// TIA Portal V17 export
// export: Created 2026-04-13T11:12:53.5499965Z, ExportSetting WithDefaults, DisplayName Totally Integrated Automation Portal, DisplayVersion V17 Update 4, DisplayName TIA Portal Openness, DisplayVersion V17 Update 4, DisplayName TIA Portal Version Control Interface, DisplayVersion V17, DisplayName SINAMICS Startdrive Advanced, DisplayVersion V17, DisplayName SINAMICS Startdrive G130, G150, S120, S150, SINAMICS MV, S210, DisplayVersion V17, DisplayName SINAMICS Startdrive G110M, G120, G120C, G120D, G120P, G115D, DisplayVersion V17, DisplayName STEP 7 Professional, DisplayVersion V17 Update 4, DisplayName STEP 7 Safety, DisplayVersion V17, DisplayName WinCC Professional, DisplayVersion V17 Update 4
TagTable "M"
  MABQ进水隔断阀 : Bool  (PLC tag MABQ进水隔断阀, HMI_连接_1, 1 s)
  MAB进水隔断阀 : Bool  (PLC tag MAB进水隔断阀, HMI_连接_1, 1 s)
  MAQ安全停机 : Bool  (PLC tag MAQ安全停机, HMI_连接_1, 1 s)
  MAS室内回水阀 : Bool  (PLC tag MAS室内回水阀, HMI_连接_1, 1 s)
  MAS室外回水阀 : Bool  (PLC tag MAS室外回水阀, HMI_连接_1, 1 s)
  MBD本地调试 : Bool  (PLC tag MBD本地调试, HMI_连接_1, 1 s)
  MBD补氮阀 : Bool  (PLC tag MBD补氮阀, HMI_连接_1, 1 s)
  MBD布袋出料 : Bool  (PLC tag MBD布袋出料, HMI_连接_1, 1 s)
  MBJ本机调试模式 : Bool  (PLC tag MBJ本机调试模式, HMI_连接_1, 1 s)
  MBS闭式进风隔断阀 : Bool  (PLC tag MBS闭式进风隔断阀, HMI_连接_1, 1 s)
  MBS闭式排风隔断阀 : Bool  (PLC tag MBS闭式排风隔断阀, HMI_连接_1, 1 s)
  MBY100 : Bool  (PLC tag MBY100, HMI_连接_1, 1 s)
  MBY101 : Bool  (PLC tag MBY101, HMI_连接_1, 1 s)
  MCC除尘出料上阀 : Bool  (PLC tag MCC除尘出料上阀, HMI_连接_1, 1 s)
  MCC除尘出料下阀 : Bool  (PLC tag MCC除尘出料下阀, HMI_连接_1, 1 s)
  MCC除尘管道清洗阀 : Bool  (PLC tag MCC除尘管道清洗阀, HMI_连接_1, 1 s)
  MCC除尘缓存震荡器 : Bool  (PLC tag MCC除尘缓存震荡器, HMI_连接_1, 1 s)
  MCC除尘脉冲 : Bool  (PLC tag MCC除尘脉冲, HMI_连接_1, 1 s)
  MCC除尘气锤 : Bool  (PLC tag MCC除尘气锤, HMI_连接_1, 1 s)
  MCC除尘清洗阀 : Bool  (PLC tag MCC除尘清洗阀, HMI_连接_1, 1 s)
  MCF出风高效清洗阀 : Bool  (PLC tag MCF出风高效清洗阀, HMI_连接_1, 1 s)
  MCS纯水洗请求 : Bool  (PLC tag MCS纯水洗请求, HMI_连接_1, 1 s)
  MCW除雾排液阀 : Bool  (PLC tag MCW除雾排液阀, HMI_连接_1, 1 s)
  MCZ初状态 : Bool  (PLC tag MCZ初状态, HMI_连接_1, 1 s)
  MDJ电加热器 : Bool  (PLC tag MDJ电加热器, HMI_连接_1, 1 s)
  MEJ二级出料 : Bool  (PLC tag MEJ二级出料, HMI_连接_1, 1 s)
  MEJ二级出料上阀 : Bool  (PLC tag MEJ二级出料上阀, HMI_连接_1, 1 s)
  MEJ二级出料下阀 : Bool  (PLC tag MEJ二级出料下阀, HMI_连接_1, 1 s)
  MEJ二级缓存震荡器 : Bool  (PLC tag MEJ二级缓存震荡器, HMI_连接_1, 1 s)
  MEJ二级冷冻水阀 : Bool  (PLC tag MEJ二级冷冻水阀, HMI_连接_1, 1 s)
  MEJ二级冷凝清洗阀 : Bool  (PLC tag MEJ二级冷凝清洗阀, HMI_连接_1, 1 s)
  MEJ二级排液阀 : Bool  (PLC tag MEJ二级排液阀, HMI_连接_1, 1 s)
  MEJ二级旋风气锤 : Bool  (PLC tag MEJ二级旋风气锤, HMI_连接_1, 1 s)
  MEJ二级旋风清洗阀 : Bool  (PLC tag MEJ二级旋风清洗阀, HMI_连接_1, 1 s)
  MEJ二级旋风振打锤 : Bool  (PLC tag MEJ二级旋风振打锤, HMI_连接_1, 1 s)
  MFK放空比例调节阀 : Bool  (PLC tag MFK放空比例调节阀, HMI_连接_1, 1 s)
  MFM蜂鸣器 : Bool  (PLC tag MFM蜂鸣器, HMI_连接_1, 1 s)
  MFZ仿真调试 : Bool  (PLC tag MFZ仿真调试, HMI_连接_1, 1 s)
  MGD管道压力手动调节 : Bool  (PLC tag MGD管道压力手动调节, HMI_连接_1, 1 s)
  MGS供水泵 : Bool  (PLC tag MGS供水泵, HMI_连接_1, 1 s)
  MHF回风加热比例调节阀 : Bool  (PLC tag MHF回风加热比例调节阀, HMI_连接_1, 1 s)
  MHF回风加热自整定 : Bool  (PLC tag MHF回风加热自整定, HMI_连接_1, 1 s)
  MHF回风温度加热 : Bool  (PLC tag MHF回风温度加热, HMI_连接_1, 1 s)
  MHF回风蒸汽开关阀 : Bool  (PLC tag MHF回风蒸汽开关阀, HMI_连接_1, 1 s)
  MHF回风蒸汽排水阀 : Bool  (PLC tag MHF回风蒸汽排水阀, HMI_连接_1, 1 s)
  MHF回风蒸汽调节阀 : Bool  (PLC tag MHF回风蒸汽调节阀, HMI_连接_1, 1 s)
  MHSQ回水隔断阀1 : Bool  (PLC tag MHSQ回水隔断阀1, HMI_连接_1, 1 s)
  MHS回水隔断阀1 : Bool  (PLC tag MHS回水隔断阀1, HMI_连接_1, 1 s)
  MJD进氮阀 : Bool  (PLC tag MJD进氮阀, HMI_连接_1, 1 s)
  MJF进风加热比例调节阀 : Bool  (PLC tag MJF进风加热比例调节阀, HMI_连接_1, 1 s)
  MJF进风冷却水阀 : Bool  (PLC tag MJF进风冷却水阀, HMI_连接_1, 1 s)
  MJF进风蒸汽比例调节阀 : Bool  (PLC tag MJF进风蒸汽比例调节阀, HMI_连接_1, 1 s)
  MJF进风蒸汽开关阀 : Bool  (PLC tag MJF进风蒸汽开关阀, HMI_连接_1, 1 s)
  MJF进风蒸汽排水阀 : Bool  (PLC tag MJF进风蒸汽排水阀, HMI_连接_1, 1 s)
  MJF进温自整定 : Bool  (PLC tag MJF进温自整定, HMI_连接_1, 1 s)
  MJL进料泵 : Bool  (PLC tag MJL进料泵, HMI_连接_1, 1 s)
  MJL进料泵风扇 : Bool  (PLC tag MJL进料泵风扇, HMI_连接_1, 1 s)
  MJL进料手动状态 : Bool  (PLC tag MJL进料手动状态, HMI_连接_1, 1 s)
  MJL进料调节 : Bool  (PLC tag MJL进料调节, HMI_连接_1, 1 s)
  MJR加热清洗阀 : Bool  (PLC tag MJR加热清洗阀, HMI_连接_1, 1 s)
  MJS碱水洗请求 : Bool  (PLC tag MJS碱水洗请求, HMI_连接_1, 1 s)
  MJS结束清洗 : Bool  (PLC tag MJS结束清洗, HMI_连接_1, 1 s)
  MJS进水调节 : Bool  (PLC tag MJS进水调节, HMI_连接_1, 1 s)
  MKS开始清洗 : Bool  (PLC tag MKS开始清洗, HMI_连接_1, 1 s)
  MKS开式进风隔断阀 : Bool  (PLC tag MKS开式进风隔断阀, HMI_连接_1, 1 s)
  MKS开式排风隔断阀 : Bool  (PLC tag MKS开式排风隔断阀, HMI_连接_1, 1 s)
  MLC料仓清洗阀 : Bool  (PLC tag MLC料仓清洗阀, HMI_连接_1, 1 s)
  MLC料仓清洗排水阀 : Bool  (PLC tag MLC料仓清洗排水阀, HMI_连接_1, 1 s)
  MLG料罐清洗阀 : Bool  (PLC tag MLG料罐清洗阀, HMI_连接_1, 1 s)
  MLS料水手动调节 : Bool  (PLC tag MLS料水手动调节, HMI_连接_1, 1 s)
  MLS料水系统调节 : Bool  (PLC tag MLS料水系统调节, HMI_连接_1, 1 s)
  MLX离心雾化 : Bool  (PLC tag MLX离心雾化, HMI_连接_1, 1 s)
  MLX离心雾化风扇 : Bool  (PLC tag MLX离心雾化风扇, HMI_连接_1, 1 s)
  MLX离心雾化油泵 : Bool  (PLC tag MLX离心雾化油泵, HMI_连接_1, 1 s)
  MMC脉冲反吹 : Bool  (PLC tag MMC脉冲反吹, HMI_连接_1, 1 s)
  MMC脉冲周期_PID : Bool  (PLC tag MMC脉冲周期_PID, HMI_连接_1, 1 s)
  MMC脉冲周期_进料 : Bool  (PLC tag MMC脉冲周期_进料, HMI_连接_1, 1 s)
  MPH平衡比例调节阀 : Bool  (PLC tag MPH平衡比例调节阀, HMI_连接_1, 1 s)
  MPS排水运行标志 : Bool  (PLC tag MPS排水运行标志, HMI_连接_1, 1 s)
  MQG气缸降 : Bool  (PLC tag MQG气缸降, HMI_连接_1, 1 s)
  MQG气缸升 : Bool  (PLC tag MQG气缸升, HMI_连接_1, 1 s)
  MQG气缸升降阀 : Bool  (PLC tag MQG气缸升降阀, HMI_连接_1, 1 s)
  MQL气流雾化阀 : Bool  (PLC tag MQL气流雾化阀, HMI_连接_1, 1 s)
  MQR确认 : Bool  (PLC tag MQR确认, HMI_连接_1, 1 s)
  MQX清洗辅助 : Bool  (PLC tag MQX清洗辅助, HMI_连接_1, 1 s)
  MQX清洗溶剂出阀 : Bool  (PLC tag MQX清洗溶剂出阀, HMI_连接_1, 1 s)
  MQX清洗溶剂罐进氮阀 : Bool  (PLC tag MQX清洗溶剂罐进氮阀, HMI_连接_1, 1 s)
  MQX清洗溶剂进阀 : Bool  (PLC tag MQX清洗溶剂进阀, HMI_连接_1, 1 s)
  MQX清洗伸缩气缸 : Bool  (PLC tag MQX清洗伸缩气缸, HMI_连接_1, 1 s)
  MQZ前置水阀 : Bool  (PLC tag MQZ前置水阀, HMI_连接_1, 1 s)
  MRC热纯加热 : Bool  (PLC tag MRC热纯加热, HMI_连接_1, 1 s)
  MRC热纯自动洗 : Bool  (PLC tag MRC热纯自动洗, HMI_连接_1, 1 s)
  MRJ溶剂回收排放阀 : Bool  (PLC tag MRJ溶剂回收排放阀, HMI_连接_1, 1 s)
  MRJ溶剂进程泵 : Bool  (PLC tag MRJ溶剂进程泵, HMI_连接_1, 1 s)
  MRJ溶剂排液泵 : Bool  (PLC tag MRJ溶剂排液泵, HMI_连接_1, 1 s)
  MRJ溶剂请求 : Bool  (PLC tag MRJ溶剂请求, HMI_连接_1, 1 s)
  MRS热水洗请求 : Bool  (PLC tag MRS热水洗请求, HMI_连接_1, 1 s)
  MSB设备振打 : Bool  (PLC tag MSB设备振打, HMI_连接_1, 1 s)
  MSC四参数关辅助 : Bool  (PLC tag MSC四参数关辅助, HMI_连接_1, 1 s)
  MSC四参数开辅助 : Bool  (PLC tag MSC四参数开辅助, HMI_连接_1, 1 s)
  MSC四参数控制 : Bool  (PLC tag MSC四参数控制, HMI_连接_1, 1 s)
  MSC四参数手动调节 : Bool  (PLC tag MSC四参数手动调节, HMI_连接_1, 1 s)
  MSC四参数手动状态 : Bool  (PLC tag MSC四参数手动状态, HMI_连接_1, 1 s)
  MSC四参数调节 : Bool  (PLC tag MSC四参数调节, HMI_连接_1, 1 s)
  MSD手动_纯水清洗 : Bool  (PLC tag MSD手动_纯水清洗, HMI_连接_1, 1 s)
  MSD手动_二纯水清洗 : Bool  (PLC tag MSD手动_二纯水清洗, HMI_连接_1, 1 s)
  MSD手动_碱水清洗 : Bool  (PLC tag MSD手动_碱水清洗, HMI_连接_1, 1 s)
  MSD手动_溶剂清洗 : Bool  (PLC tag MSD手动_溶剂清洗, HMI_连接_1, 1 s)
  MSD手动_溶剂清洗(1) : Bool  (PLC tag "MSD手动_溶剂清洗(1)", HMI_连接_1, 1 s)
  MSF输送风机 : Bool  (PLC tag MSF输送风机, HMI_连接_1, 1 s)
  MSF输送加热器 : Bool  (PLC tag MSF输送加热器, HMI_连接_1, 1 s)
  MSF送风机 : Bool  (PLC tag MSF送风机, HMI_连接_1, 1 s)
  MSF送风机风扇 : Bool  (PLC tag MSF送风机风扇, HMI_连接_1, 1 s)
  MSF送风机排水阀 : Bool  (PLC tag MSF送风机排水阀, HMI_连接_1, 1 s)
  MSF送风机清洗阀 : Bool  (PLC tag MSF送风机清洗阀, HMI_连接_1, 1 s)
  MSJ水进程泵 : Bool  (PLC tag MSJ水进程泵, HMI_连接_1, 1 s)
  MSN室内排水隔膜泵 : Bool  (PLC tag MSN室内排水隔膜泵, HMI_连接_1, 1 s)
  MSN室内清洗总阀 : Bool  (PLC tag MSN室内清洗总阀, HMI_连接_1, 1 s)
  MSS输送出料 : Bool  (PLC tag MSS输送出料, HMI_连接_1, 1 s)
  MSS输送出料上阀 : Bool  (PLC tag MSS输送出料上阀, HMI_连接_1, 1 s)
  MSS输送出料下阀 : Bool  (PLC tag MSS输送出料下阀, HMI_连接_1, 1 s)
  MSS输送管路排水阀 : Bool  (PLC tag MSS输送管路排水阀, HMI_连接_1, 1 s)
  MSS输送管路清洗阀 : Bool  (PLC tag MSS输送管路清洗阀, HMI_连接_1, 1 s)
  MSS输送加热 : Bool  (PLC tag MSS输送加热, HMI_连接_1, 1 s)
  MSS输送进风阀 : Bool  (PLC tag MSS输送进风阀, HMI_连接_1, 1 s)
  MSS输送系统 : Bool  (PLC tag MSS输送系统, HMI_连接_1, 1 s)
  MSS输送自整定 : Bool  (PLC tag MSS输送自整定, HMI_连接_1, 1 s)
  MTD塔顶清洗球阀 : Bool  (PLC tag MTD塔顶清洗球阀, HMI_连接_1, 1 s)
  MWK蜗壳清洗阀 : Bool  (PLC tag MWK蜗壳清洗阀, HMI_连接_1, 1 s)
  MWL物料进阀 : Bool  (PLC tag MWL物料进阀, HMI_连接_1, 1 s)
  MXF旋风管道清洗阀 : Bool  (PLC tag MXF旋风管道清洗阀, HMI_连接_1, 1 s)
  MXT心跳接受信号 : Bool  (PLC tag MXT心跳接受信号, HMI_连接_1, 1 s)
  MXY泄压阀 : Bool  (PLC tag MXY泄压阀, HMI_连接_1, 1 s)
  MXY泄压请求 : Bool  (PLC tag MXY泄压请求, HMI_连接_1, 1 s)
  MYF引风机 : Bool  (PLC tag MYF引风机, HMI_连接_1, 1 s)
  MYF引风机风扇 : Bool  (PLC tag MYF引风机风扇, HMI_连接_1, 1 s)
  MYF引风机排水阀 : Bool  (PLC tag MYF引风机排水阀, HMI_连接_1, 1 s)
  MYF引风机清洗阀 : Bool  (PLC tag MYF引风机清洗阀, HMI_连接_1, 1 s)
  MYG压干请求 : Bool  (PLC tag MYG压干请求, HMI_连接_1, 1 s)
  MYH氧含仪隔断阀 : Bool  (PLC tag MYH氧含仪隔断阀, HMI_连接_1, 1 s)
  MYJ二级冷冻水阀 : Bool  (PLC tag MYJ二级冷冻水阀, HMI_连接_1, 1 s)
  MYJ一级出料 : Bool  (PLC tag MYJ一级出料, HMI_连接_1, 1 s)
  MYJ一级出料上阀 : Bool  (PLC tag MYJ一级出料上阀, HMI_连接_1, 1 s)
  MYJ一级出料下阀 : Bool  (PLC tag MYJ一级出料下阀, HMI_连接_1, 1 s)
  MYJ一级缓存振荡器 : Bool  (PLC tag MYJ一级缓存振荡器, HMI_连接_1, 1 s)
  MYJ一级冷凝清洗阀 : Bool  (PLC tag MYJ一级冷凝清洗阀, HMI_连接_1, 1 s)
  MYJ一级冷却水阀 : Bool  (PLC tag MYJ一级冷却水阀, HMI_连接_1, 1 s)
  MYJ一级排液阀 : Bool  (PLC tag MYJ一级排液阀, HMI_连接_1, 1 s)
  MYJ一级旋风气锤 : Bool  (PLC tag MYJ一级旋风气锤, HMI_连接_1, 1 s)
  MYJ一级旋风清洗阀 : Bool  (PLC tag MYJ一级旋风清洗阀, HMI_连接_1, 1 s)
  MYJ一级旋风振打锤 : Bool  (PLC tag MYJ一级旋风振打锤, HMI_连接_1, 1 s)
  MYJ一级旋风振荡器 : Bool  (PLC tag MYJ一级旋风振荡器, HMI_连接_1, 1 s)
  MYS钥匙开关 : Bool  (PLC tag MYS钥匙开关, HMI_连接_1, 1 s)
  MZB准备清洗 : Bool  (PLC tag MZB准备清洗, HMI_连接_1, 1 s)
  MZD自动清洗 : Bool  (PLC tag MZD自动清洗, HMI_连接_1, 1 s)
  MZS指示灯 : Bool  (PLC tag MZS指示灯, HMI_连接_1, 1 s)
  MZS注射水请求 : Bool  (PLC tag MZS注射水请求, HMI_连接_1, 1 s)
  MZT暂停辅助 : Bool  (PLC tag MZT暂停辅助, HMI_连接_1, 1 s)
  MZT主塔排水阀 : Bool  (PLC tag MZT主塔排水阀, HMI_连接_1, 1 s)
  MZT主塔气锤 : Bool  (PLC tag MZT主塔气锤, HMI_连接_1, 1 s)
  MZT主塔清洗 : Bool  (PLC tag MZT主塔清洗, HMI_连接_1, 1 s)
  MZT主塔清洗进水阀 : Bool  (PLC tag MZT主塔清洗进水阀, HMI_连接_1, 1 s)
  MZT主塔伸缩气缸 : Bool  (PLC tag MZT主塔伸缩气缸, HMI_连接_1, 1 s)
  MZT总通路 : Bool  (PLC tag MZT总通路, HMI_连接_1, 1 s)
  QXY泄压请求 : Bool  (PLC tag QXY泄压请求, HMI_连接_1, 1 s)
